TYPE EM_Transport_Mechanische_Stop_CS :
STRUCT
	Start		: BOOL;
	Stop		: BOOL;
	Reset		: BOOL;
	Abort		: BOOL;
	Auto		: BOOL;
	Manueel		: BOOL;
END_STRUCT
END_TYPE

(* stored: Version 1.1.0.1, ProductVersion 3.1.4024.12
   DUT EM_Transport_Mechanische_Stop_CS: Id {8713c655-a17c-45e9-8ef9-a7c88d017419} *)
